Fanuc KAREL source: VREG_OFFSET.kl

PROGRAM T
%NOLOCKGROUP
VAR
 v0 : INTEGER
 v1 : INTEGER
 v2 : INTEGER
BEGIN
 VREG_OFFSET(v0, v1, v2)
END T
